// TwinCAT 3 PLC project LAP_2010_2_Transportwagen
// ProgramVersion: 3.1.4022.1
// libraries:
//   Tc2_Standard, * (Beckhoff Automation GmbH)
//   Tc2_System, * (Beckhoff Automation GmbH)
//   Tc2_Utilities, * (Beckhoff Automation GmbH)
//   Tc3_Module, * (Beckhoff Automation GmbH)
// project tree:
//   GVLs/ PlcCx9020.TcGVL, SimDI.TcGVL, SimDA.TcGVL, DigInput.TcGVL (not stored), DigOutput.TcGVL (not stored), AnalogInput.TcGVL (not stored), AnalogOutput.TcGVL (not stored), VersionsInfo.TcGVL (not stored)
//   / PlcTask.TcTTO (not stored)
//   POUs/ MAIN.TcPOU, Transportwagen.TcPOU
//   POUs/Privat/ AlleBitSetzen.TcPOU (not stored), BitLesen.TcPOU (not stored), DatenRangieren.TcPOU
// real-time tasks:
//   TASK PlcTask: cycle T#10ms, priority 20, ADS port 350
// motion (NC):
//   TASK NC-Task 1 SAF: cycle T#2ms, priority 4, ADS port 501
//   TASK NC-Task 1 SVB: cycle T#10ms, priority 8, ADS port 511
//   AXIS Axis 1 (id 1)
//     OtherSettings: AllowMotionCmdToSlave=true
//     encoder EncType=4
//       EncPara: MaxCount=#x0000ffff
//         Inc: RefSoftSyncMask=#x0000ffff
//     drive DrvType=24
//       Analog: ScaleFactorActTorque=0.1
//       TimeComp: TaskDelayCycles=1
//     controller CtrType=1
//       CtrPara: PriorControlFactor=1
//         Observer: BandWidth=20
//   AXIS Axis 2 (id 2)
//     OtherSettings: AllowMotionCmdToSlave=true
//     encoder EncType=4
//       EncPara: MaxCount=#x0000ffff
//         Inc: RefSoftSyncMask=#x0000ffff
//     drive DrvType=24
//       Analog: ScaleFactorActTorque=0.1
//       TimeComp: TaskDelayCycles=1
//     controller CtrType=1
//       CtrPara: PriorControlFactor=1
//         Observer: BandWidth=20
//   AXIS Axis 3 (id 3)
//     OtherSettings: AllowMotionCmdToSlave=true
//     encoder EncType=4
//       EncPara: MaxCount=#x0000ffff
//     drive DrvType=23
//       Analog: ScaleFactorActTorque=0.1
//       TimeComp: TaskDelayCycles=1
//     controller CtrType=1
//       CtrPara: PriorControlFactor=1
//         Observer: BandWidth=20
//   AXIS Axis 4 (id 4)
//     OtherSettings: AllowMotionCmdToSlave=true
//     encoder EncType=4
//       EncPara: MaxCount=#x0000ffff
//     drive DrvType=23
//       Analog: ScaleFactorActTorque=0.1
//       TimeComp: TaskDelayCycles=1
//     controller CtrType=1
//       CtrPara: PriorControlFactor=1
//         Observer: BandWidth=20
//   AXIS Axis 5 (id 5)
//     OtherSettings: AllowMotionCmdToSlave=true
//     encoder EncType=19
//       EncPara: MaxCount=#xffffffff
//     drive DrvType=16
//       DrvPara: MaxCount=#xffffffff
//         Analog: ScaleFactorActTorque=0.1
//         TimeComp: TaskDelayCycles=1
//     controller CtrType=1
//       CtrPara: PriorControlFactor=1
//         Observer: BandWidth=20
//   AXIS Axis 6 (id 6)
//     OtherSettings: AllowMotionCmdToSlave=true
//     encoder EncType=19
//       EncPara: MaxCount=#xffffffff
//     drive DrvType=16
//       DrvPara: MaxCount=#xffffffff
//         Analog: ScaleFactorActTorque=0.1
//         TimeComp: TaskDelayCycles=1
//     controller CtrType=1
//       CtrPara: PriorControlFactor=1
//         Observer: BandWidth=20
// I/O:
//   DEVICE Device 1 (EtherCAT), AmsNetId 192.168.0.200.2.1
//     Term 1 (EK1200) [EK1200-5000 EtherCAT Power supply (2A E-Bus)]
//       Term 2 (EL1809) [EL1809 16Ch. Dig. Input 24V, 3ms]
//       Term 3 (EL1809) [EL1809 16Ch. Dig. Input 24V, 3ms]
//       Term 4 (EL2809) [EL2809 16Ch. Dig. Output 24V, 0.5A]
//       Term 5 (EL2809) [EL2809 16Ch. Dig. Output 24V, 0.5A]
//       Term 6 (EL3064) [EL3064 4Ch. Ana. Input 0-10V]
//       Term 7 (EL4034) [EL4034 4Ch. Ana. Output +/-10V, 12bit]
//       Term 8 (EL7031) [EL7031 1Ch. Stepper motor output stage (24V, 1.5A)]
//       Term 9 (EL7031) [EL7031 1Ch. Stepper motor output stage (24V, 1.5A)]
//       Term 10 (EL7332) [EL7332 2Ch. DC motor output stage (24V, 1.5A)]
//       Term 11 (EL7201-0010) [EL7201-0010 1Ch. MDP742 Servo motor output stage with OCT (50V, 4A)]
//       Term 12 (EL7201-0010) [EL7201-0010 1Ch. MDP742 Servo motor output stage with OCT (50V, 4A)]
//       Term 26 (EL6090) [EL6090 Display terminal]
//       Term 27 (EK1110) [EK1110 EtherCAT extension]
// variable links:
//   NC-Task 1 SAF/Axes/Axis 1 <-> Device 1 (EtherCAT)/Term 1 (EK1200)/Term 8 (EL7031)
//     Drive/Inputs/In/nState1 @bit 3 <-> STM Status/Status/Error
//     Drive/Inputs/In/nState1 @bit 5 <-> STM Status/Status/Moving negative
//     Drive/Inputs/In/nState1 @bit 4 <-> STM Status/Status/Moving positive
//     Drive/Inputs/In/nState1 @bit 1 <-> STM Status/Status/Ready
//     Drive/Inputs/In/nState1 <-> STM Status/Status/Ready to enable
//     Drive/Inputs/In/nState1 @bit 6 <-> STM Status/Status/Torque reduced
//     Drive/Inputs/In/nState1 @bit 2 <-> STM Status/Status/Warning
//     Drive/Inputs/In/nState2 @bit 3 <-> STM Status/Status/Digital input 1
//     Drive/Inputs/In/nState2 @bit 4 <-> STM Status/Status/Digital input 2
//     Drive/Inputs/In/nState2 @bit 5 <-> STM Status/Status/Sync error
//     Drive/Inputs/In/nState2 @bit 7 <-> STM Status/Status/TxPDO Toggle
//     Drive/Inputs/In/nState4 @bit 1 <-> WcState/InputToggle
//     Drive/Inputs/In/nState4 <-> WcState/WcState
//     Drive/Outputs/Out/nCtrl1 <-> STM Control/Control/Enable
//     Drive/Outputs/Out/nCtrl1 @bit 2 <-> STM Control/Control/Reduce torque
//     Drive/Outputs/Out/nCtrl1 @bit 1 <-> STM Control/Control/Reset
//     Drive/Outputs/Out/nDataOut2[0] <-> STM Velocity/Velocity
//     Enc/Inputs/In/nDataIn1[0] <-> ENC Status compact/Counter value
//     Enc/Inputs/In/nDataIn2[0] <-> ENC Status compact/Latch value
//     Enc/Inputs/In/nState1 @bit 4 <-> ENC Status compact/Status/Counter overflow
//     Enc/Inputs/In/nState1 @bit 3 <-> ENC Status compact/Status/Counter underflow
//     Enc/Inputs/In/nState1 @bit 1 <-> ENC Status compact/Status/Latch extern valid
//     Enc/Inputs/In/nState1 @bit 2 <-> ENC Status compact/Status/Set counter done
//     Enc/Inputs/In/nState2 @bit 4 <-> ENC Status compact/Status/Status of extern latch
//     Enc/Inputs/In/nState2 @bit 5 <-> ENC Status compact/Status/Sync error
//     Enc/Inputs/In/nState2 @bit 7 <-> ENC Status compact/Status/TxPDO Toggle
//     Enc/Inputs/In/nState4 @bit 1 <-> WcState/InputToggle
//     Enc/Inputs/In/nState4 <-> WcState/WcState
//     Enc/Outputs/Out/nCtrl1 @bit 3 <-> ENC Control compact/Control/Enable latch extern on negative edge
//     Enc/Outputs/Out/nCtrl1 @bit 1 <-> ENC Control compact/Control/Enable latch extern on positive edge
//     Enc/Outputs/Out/nCtrl1 @bit 2 <-> ENC Control compact/Control/Set counter
//     Enc/Outputs/Out/nDataOut1[0] <-> ENC Control compact/Set counter value
//   NC-Task 1 SAF/Axes/Axis 2 <-> Device 1 (EtherCAT)/Term 1 (EK1200)/Term 9 (EL7031)
//     Drive/Inputs/In/nState1 @bit 3 <-> STM Status/Status/Error
//     Drive/Inputs/In/nState1 @bit 5 <-> STM Status/Status/Moving negative
//     Drive/Inputs/In/nState1 @bit 4 <-> STM Status/Status/Moving positive
//     Drive/Inputs/In/nState1 @bit 1 <-> STM Status/Status/Ready
//     Drive/Inputs/In/nState1 <-> STM Status/Status/Ready to enable
//     Drive/Inputs/In/nState1 @bit 6 <-> STM Status/Status/Torque reduced
//     Drive/Inputs/In/nState1 @bit 2 <-> STM Status/Status/Warning
//     Drive/Inputs/In/nState2 @bit 3 <-> STM Status/Status/Digital input 1
//     Drive/Inputs/In/nState2 @bit 4 <-> STM Status/Status/Digital input 2
//     Drive/Inputs/In/nState2 @bit 5 <-> STM Status/Status/Sync error
//     Drive/Inputs/In/nState2 @bit 7 <-> STM Status/Status/TxPDO Toggle
//     Drive/Inputs/In/nState4 @bit 1 <-> WcState/InputToggle
//     Drive/Inputs/In/nState4 <-> WcState/WcState
//     Drive/Outputs/Out/nCtrl1 <-> STM Control/Control/Enable
//     Drive/Outputs/Out/nCtrl1 @bit 2 <-> STM Control/Control/Reduce torque
//     Drive/Outputs/Out/nCtrl1 @bit 1 <-> STM Control/Control/Reset
//     Drive/Outputs/Out/nDataOut2[0] <-> STM Velocity/Velocity
//     Enc/Inputs/In/nDataIn1[0] <-> ENC Status compact/Counter value
//     Enc/Inputs/In/nDataIn2[0] <-> ENC Status compact/Latch value
//     Enc/Inputs/In/nState1 @bit 4 <-> ENC Status compact/Status/Counter overflow
//     Enc/Inputs/In/nState1 @bit 3 <-> ENC Status compact/Status/Counter underflow
//     Enc/Inputs/In/nState1 @bit 1 <-> ENC Status compact/Status/Latch extern valid
//     Enc/Inputs/In/nState1 @bit 2 <-> ENC Status compact/Status/Set counter done
//     Enc/Inputs/In/nState2 @bit 4 <-> ENC Status compact/Status/Status of extern latch
//     Enc/Inputs/In/nState2 @bit 5 <-> ENC Status compact/Status/Sync error
//     Enc/Inputs/In/nState2 @bit 7 <-> ENC Status compact/Status/TxPDO Toggle
//     Enc/Inputs/In/nState4 @bit 1 <-> WcState/InputToggle
//     Enc/Inputs/In/nState4 <-> WcState/WcState
//     Enc/Outputs/Out/nCtrl1 @bit 3 <-> ENC Control compact/Control/Enable latch extern on negative edge
//     Enc/Outputs/Out/nCtrl1 @bit 1 <-> ENC Control compact/Control/Enable latch extern on positive edge
//     Enc/Outputs/Out/nCtrl1 @bit 2 <-> ENC Control compact/Control/Set counter
//     Enc/Outputs/Out/nDataOut1[0] <-> ENC Control compact/Set counter value
//   NC-Task 1 SAF/Axes/Axis 3 <-> Device 1 (EtherCAT)/Term 1 (EK1200)/Term 10 (EL7332)
//     Drive/Inputs/In/nState1 @bit 3 <-> DCM Status Channel 1/Status/Error
//     Drive/Inputs/In/nState1 @bit 5 <-> DCM Status Channel 1/Status/Moving negative
//     Drive/Inputs/In/nState1 @bit 4 <-> DCM Status Channel 1/Status/Moving positive
//     Drive/Inputs/In/nState1 @bit 1 <-> DCM Status Channel 1/Status/Ready
//     Drive/Inputs/In/nState1 <-> DCM Status Channel 1/Status/Ready to enable
//     Drive/Inputs/In/nState1 @bit 6 <-> DCM Status Channel 1/Status/Torque reduced
//     Drive/Inputs/In/nState1 @bit 2 <-> DCM Status Channel 1/Status/Warning
//     Drive/Inputs/In/nState2 @bit 3 <-> DCM Status Channel 1/Status/Digital input 1
//     Drive/Inputs/In/nState2 @bit 4 <-> DCM Status Channel 1/Status/Digital input 2
//     Drive/Inputs/In/nState2 @bit 5 <-> DCM Status Channel 1/Status/Sync error
//     Drive/Inputs/In/nState2 @bit 7 <-> DCM Status Channel 1/Status/TxPDO Toggle
//     Drive/Inputs/In/nState4 @bit 1 <-> WcState/InputToggle
//     Drive/Inputs/In/nState4 <-> WcState/WcState
//     Drive/Outputs/Out/nCtrl1 <-> DCM Control Channel 1/Control/Enable
//     Drive/Outputs/Out/nCtrl1 @bit 2 <-> DCM Control Channel 1/Control/Reduce torque
//     Drive/Outputs/Out/nCtrl1 @bit 1 <-> DCM Control Channel 1/Control/Reset
//     Drive/Outputs/Out/nDataOut2[0] <-> DCM Velocity Channel 1/Velocity
//   NC-Task 1 SAF/Axes/Axis 4 <-> Device 1 (EtherCAT)/Term 1 (EK1200)/Term 10 (EL7332)
//     Drive/Inputs/In/nState1 @bit 3 <-> DCM Status Channel 2/Status/Error
//     Drive/Inputs/In/nState1 @bit 5 <-> DCM Status Channel 2/Status/Moving negative
//     Drive/Inputs/In/nState1 @bit 4 <-> DCM Status Channel 2/Status/Moving positive
//     Drive/Inputs/In/nState1 @bit 1 <-> DCM Status Channel 2/Status/Ready
//     Drive/Inputs/In/nState1 <-> DCM Status Channel 2/Status/Ready to enable
//     Drive/Inputs/In/nState1 @bit 6 <-> DCM Status Channel 2/Status/Torque reduced
//     Drive/Inputs/In/nState1 @bit 2 <-> DCM Status Channel 2/Status/Warning
//     Drive/Inputs/In/nState2 @bit 3 <-> DCM Status Channel 2/Status/Digital input 1
//     Drive/Inputs/In/nState2 @bit 4 <-> DCM Status Channel 2/Status/Digital input 2
//     Drive/Inputs/In/nState2 @bit 5 <-> DCM Status Channel 2/Status/Sync error
//     Drive/Inputs/In/nState2 @bit 7 <-> DCM Status Channel 2/Status/TxPDO Toggle
//     Drive/Inputs/In/nState4 @bit 1 <-> WcState/InputToggle
//     Drive/Inputs/In/nState4 <-> WcState/WcState
//     Drive/Outputs/Out/nCtrl1 <-> DCM Control Channel 2/Control/Enable
//     Drive/Outputs/Out/nCtrl1 @bit 2 <-> DCM Control Channel 2/Control/Reduce torque
//     Drive/Outputs/Out/nCtrl1 @bit 1 <-> DCM Control Channel 2/Control/Reset
//     Drive/Outputs/Out/nDataOut2[0] <-> DCM Velocity Channel 2/Velocity
//   NC-Task 1 SAF/Axes/Axis 5 <-> Device 1 (EtherCAT)/Term 1 (EK1200)/Term 11 (EL7201-0010)
//     Drive/Inputs/In/nDcOutputTime <-> InfoData/DcOutputShift
//     Drive/Inputs/In/nState1 <-> DRV Statusword/Statusword
//     Drive/Inputs/In/nState2 <-> DRV Statusword/Statusword @bit 8
//     Drive/Inputs/In/nState4 @bit 1 <-> WcState/InputToggle
//     Drive/Inputs/In/nState4 <-> WcState/WcState
//     Drive/Outputs/Out/nCtrl1 <-> DRV Controlword/Controlword
//     Drive/Outputs/Out/nCtrl2 <-> DRV Controlword/Controlword @bit 8
//     Drive/Outputs/Out/nDataOut2 <-> DRV Target velocity/Target velocity
//     Enc/Inputs/In/nDataIn1 <-> FB Position/Position
//     Enc/Inputs/In/nDcInputTime <-> InfoData/DcInputShift
//     Enc/Inputs/In/nState4 @bit 1 <-> WcState/InputToggle
//     Enc/Inputs/In/nState4 <-> WcState/WcState
//   NC-Task 1 SAF/Axes/Axis 6 <-> Device 1 (EtherCAT)/Term 1 (EK1200)/Term 12 (EL7201-0010)
//     Drive/Inputs/In/nDcOutputTime <-> InfoData/DcOutputShift
//     Drive/Inputs/In/nState1 <-> DRV Statusword/Statusword
//     Drive/Inputs/In/nState2 <-> DRV Statusword/Statusword @bit 8
//     Drive/Inputs/In/nState4 @bit 1 <-> WcState/InputToggle
//     Drive/Inputs/In/nState4 <-> WcState/WcState
//     Drive/Outputs/Out/nCtrl1 <-> DRV Controlword/Controlword
//     Drive/Outputs/Out/nCtrl2 <-> DRV Controlword/Controlword @bit 8
//     Drive/Outputs/Out/nDataOut2 <-> DRV Target velocity/Target velocity
//     Enc/Inputs/In/nDataIn1 <-> FB Position/Position
//     Enc/Inputs/In/nDcInputTime <-> InfoData/DcInputShift
//     Enc/Inputs/In/nState4 @bit 1 <-> WcState/InputToggle
//     Enc/Inputs/In/nState4 <-> WcState/WcState
//   LAP_2010_2_Transportwagen/LAP_2010_2_Transportwagen Instance <-> Device 1 (EtherCAT)/Term 1 (EK1200)/Term 2 (EL1809)
//     PlcTask Inputs/PlcCx9020.DI_0_0 <-> Channel 1/Input
//     PlcTask Inputs/PlcCx9020.DI_0_1 <-> Channel 2/Input
//     PlcTask Inputs/PlcCx9020.DI_0_2 <-> Channel 3/Input
//     PlcTask Inputs/PlcCx9020.DI_0_3 <-> Channel 4/Input
//     PlcTask Inputs/PlcCx9020.DI_0_4 <-> Channel 5/Input
//     PlcTask Inputs/PlcCx9020.DI_0_5 <-> Channel 6/Input
//     PlcTask Inputs/PlcCx9020.DI_0_6 <-> Channel 7/Input
//     PlcTask Inputs/PlcCx9020.DI_0_7 <-> Channel 8/Input
//     PlcTask Inputs/PlcCx9020.DI_1_0 <-> Channel 9/Input
//     PlcTask Inputs/PlcCx9020.DI_1_1 <-> Channel 10/Input
//     PlcTask Inputs/PlcCx9020.DI_1_2 <-> Channel 11/Input
//     PlcTask Inputs/PlcCx9020.DI_1_3 <-> Channel 12/Input
//     PlcTask Inputs/PlcCx9020.DI_1_4 <-> Channel 13/Input
//     PlcTask Inputs/PlcCx9020.DI_1_5 <-> Channel 14/Input
//     PlcTask Inputs/PlcCx9020.DI_1_6 <-> Channel 15/Input
//     PlcTask Inputs/PlcCx9020.DI_1_7 <-> Channel 16/Input
//   LAP_2010_2_Transportwagen/LAP_2010_2_Transportwagen Instance <-> Device 1 (EtherCAT)/Term 1 (EK1200)/Term 3 (EL1809)
//     PlcTask Inputs/PlcCx9020.DI_2_0 <-> Channel 1/Input
//     PlcTask Inputs/PlcCx9020.DI_2_1 <-> Channel 2/Input
//     PlcTask Inputs/PlcCx9020.DI_2_2 <-> Channel 3/Input
//     PlcTask Inputs/PlcCx9020.DI_2_3 <-> Channel 4/Input
//     PlcTask Inputs/PlcCx9020.DI_2_4 <-> Channel 5/Input
//     PlcTask Inputs/PlcCx9020.DI_2_5 <-> Channel 6/Input
//     PlcTask Inputs/PlcCx9020.DI_2_6 <-> Channel 7/Input
//     PlcTask Inputs/PlcCx9020.DI_2_7 <-> Channel 8/Input
//     PlcTask Inputs/PlcCx9020.DI_3_0 <-> Channel 9/Input
//     PlcTask Inputs/PlcCx9020.DI_3_1 <-> Channel 10/Input
//     PlcTask Inputs/PlcCx9020.DI_3_2 <-> Channel 11/Input
//     PlcTask Inputs/PlcCx9020.DI_3_3 <-> Channel 12/Input
//     PlcTask Inputs/PlcCx9020.DI_3_4 <-> Channel 13/Input
//     PlcTask Inputs/PlcCx9020.DI_3_5 <-> Channel 14/Input
//     PlcTask Inputs/PlcCx9020.DI_3_6 <-> Channel 15/Input
//     PlcTask Inputs/PlcCx9020.DI_3_7 <-> Channel 16/Input
//   LAP_2010_2_Transportwagen/LAP_2010_2_Transportwagen Instance <-> Device 1 (EtherCAT)/Term 1 (EK1200)/Term 4 (EL2809)
//     PlcTask Outputs/PlcCx9020.DA_0_0 <-> Channel 1/Output
//     PlcTask Outputs/PlcCx9020.DA_0_1 <-> Channel 2/Output
//     PlcTask Outputs/PlcCx9020.DA_0_2 <-> Channel 3/Output
//     PlcTask Outputs/PlcCx9020.DA_0_3 <-> Channel 4/Output
//     PlcTask Outputs/PlcCx9020.DA_0_4 <-> Channel 5/Output
//     PlcTask Outputs/PlcCx9020.DA_0_5 <-> Channel 6/Output
//     PlcTask Outputs/PlcCx9020.DA_0_6 <-> Channel 7/Output
//     PlcTask Outputs/PlcCx9020.DA_0_7 <-> Channel 8/Output
//     PlcTask Outputs/PlcCx9020.DA_1_0 <-> Channel 9/Output
//     PlcTask Outputs/PlcCx9020.DA_1_1 <-> Channel 10/Output
//     PlcTask Outputs/PlcCx9020.DA_1_2 <-> Channel 11/Output
//     PlcTask Outputs/PlcCx9020.DA_1_3 <-> Channel 12/Output
//     PlcTask Outputs/PlcCx9020.DA_1_4 <-> Channel 13/Output
//     PlcTask Outputs/PlcCx9020.DA_1_5 <-> Channel 14/Output
//     PlcTask Outputs/PlcCx9020.DA_1_6 <-> Channel 15/Output
//     PlcTask Outputs/PlcCx9020.DA_1_7 <-> Channel 16/Output
//   LAP_2010_2_Transportwagen/LAP_2010_2_Transportwagen Instance <-> Device 1 (EtherCAT)/Term 1 (EK1200)/Term 5 (EL2809)
//     PlcTask Outputs/PlcCx9020.DA_2_0 <-> Channel 1/Output
//     PlcTask Outputs/PlcCx9020.DA_2_1 <-> Channel 2/Output
//     PlcTask Outputs/PlcCx9020.DA_2_2 <-> Channel 3/Output
//     PlcTask Outputs/PlcCx9020.DA_2_3 <-> Channel 4/Output
//     PlcTask Outputs/PlcCx9020.DA_2_4 <-> Channel 5/Output
//     PlcTask Outputs/PlcCx9020.DA_2_5 <-> Channel 6/Output
//     PlcTask Outputs/PlcCx9020.DA_2_6 <-> Channel 7/Output
//     PlcTask Outputs/PlcCx9020.DA_2_7 <-> Channel 8/Output
//     PlcTask Outputs/PlcCx9020.DA_3_0 <-> Channel 9/Output
//     PlcTask Outputs/PlcCx9020.DA_3_1 <-> Channel 10/Output
//     PlcTask Outputs/PlcCx9020.DA_3_2 <-> Channel 11/Output
//     PlcTask Outputs/PlcCx9020.DA_3_3 <-> Channel 12/Output
//     PlcTask Outputs/PlcCx9020.DA_3_4 <-> Channel 13/Output
//     PlcTask Outputs/PlcCx9020.DA_3_5 <-> Channel 14/Output
//     PlcTask Outputs/PlcCx9020.DA_3_6 <-> Channel 15/Output
//     PlcTask Outputs/PlcCx9020.DA_3_7 <-> Channel 16/Output
//   LAP_2010_2_Transportwagen/LAP_2010_2_Transportwagen Instance <-> Device 1 (EtherCAT)/Term 1 (EK1200)/Term 6 (EL3064)
//     PlcTask Inputs/PlcCx9020.AI_{0..3} <-> AI Standard Channel {1..4}/Value  (4 links)
//   LAP_2010_2_Transportwagen/LAP_2010_2_Transportwagen Instance <-> Device 1 (EtherCAT)/Term 1 (EK1200)/Term 7 (EL4034)
//     PlcTask Outputs/PlcCx9020.AA_{0..3} <-> AO Outputs Channel {1..4}/Analog output  (4 links)

// ---- GVLs/PlcCx9020.TcGVL
{attribute 'qualified_only'}
VAR_GLOBAL
	// dSub 25
	DI_0_0 AT %IX0.0: BOOL;
	DI_0_1 AT %IX0.1: BOOL;
	DI_0_2 AT %IX0.2: BOOL;
	DI_0_3 AT %IX0.3: BOOL;
	DI_0_4 AT %IX0.4: BOOL;
	DI_0_5 AT %IX0.5: BOOL;
	DI_0_6 AT %IX0.6: BOOL;
	DI_0_7 AT %IX0.7: BOOL;
	DI_1_0 AT %IX1.0: BOOL;
	DI_1_1 AT %IX1.1: BOOL;
	DI_1_2 AT %IX1.2: BOOL;
	DI_1_3 AT %IX1.3: BOOL;
	DI_1_4 AT %IX1.4: BOOL;
	DI_1_5 AT %IX1.5: BOOL;
	DI_1_6 AT %IX1.6: BOOL;
	DI_1_7 AT %IX1.7: BOOL;
	// Sicherheitsbuchsen
	DI_2_0 AT %IX2.0: BOOL;
	DI_2_1 AT %IX2.1: BOOL;
	DI_2_2 AT %IX2.2: BOOL;
	DI_2_3 AT %IX2.3: BOOL;
	DI_2_4 AT %IX2.4: BOOL;
	DI_2_5 AT %IX2.5: BOOL;
	DI_2_6 AT %IX2.6: BOOL;
	DI_2_7 AT %IX2.7: BOOL;
	DI_3_0 AT %IX3.0: BOOL;
	DI_3_1 AT %IX3.1: BOOL;
	DI_3_2 AT %IX3.2: BOOL;
	DI_3_3 AT %IX3.3: BOOL;
	DI_3_4 AT %IX3.4: BOOL;
	DI_3_5 AT %IX3.5: BOOL;
	DI_3_6 AT %IX3.6: BOOL;
	DI_3_7 AT %IX3.7: BOOL;
	DI AT %IB0: ARRAY[0..3] OF BYTE; 

	// dSub 25
	DA_0_0 AT %QX0.0: BOOL;
	DA_0_1 AT %QX0.1: BOOL;
	DA_0_2 AT %QX0.2: BOOL;
	DA_0_3 AT %QX0.3: BOOL;
	DA_0_4 AT %QX0.4: BOOL;
	DA_0_5 AT %QX0.5: BOOL;
	DA_0_6 AT %QX0.6: BOOL;
	DA_0_7 AT %QX0.7: BOOL;
	DA_1_0 AT %QX1.0: BOOL;
	DA_1_1 AT %QX1.1: BOOL;
	DA_1_2 AT %QX1.2: BOOL;
	DA_1_3 AT %QX1.3: BOOL;
	DA_1_4 AT %QX1.4: BOOL;
	DA_1_5 AT %QX1.5: BOOL;
	DA_1_6 AT %QX1.6: BOOL;
	DA_1_7 AT %QX1.7: BOOL;
	// Sicherheitsbuchsen
	DA_2_0 AT %QX2.0: BOOL;
	DA_2_1 AT %QX2.1: BOOL;
	DA_2_2 AT %QX2.2: BOOL;
	DA_2_3 AT %QX2.3: BOOL;
	DA_2_4 AT %QX2.4: BOOL;
	DA_2_5 AT %QX2.5: BOOL;
	DA_2_6 AT %QX2.6: BOOL;
	DA_2_7 AT %QX2.7: BOOL;
	DA_3_0 AT %QX3.0: BOOL;
	DA_3_1 AT %QX3.1: BOOL;
	DA_3_2 AT %QX3.2: BOOL;
	DA_3_3 AT %QX3.3: BOOL;
	DA_3_4 AT %QX3.4: BOOL;
	DA_3_5 AT %QX3.5: BOOL;
	DA_3_6 AT %QX3.6: BOOL;
	DA_3_7 AT %QX3.7: BOOL;
	DA AT %QB0: ARRAY[0..3] OF BYTE;
	
	// dSub 25
	AI_0 AT %IW10: INT;			// Analogeingang 0
	AI_1 AT %IW12: INT;			// Analogeingang 1
	
	// Sicherheitsbuchsen
	AI_2 AT %IW14: INT;			// Analogeingang 2
	AI_3 AT %IW16: INT;			// Analogeingang 3
	AI AT %IW10: ARRAY[0..7] OF BYTE;
	
	
	// dSub 25
	AA_0 AT %QW10: INT;			// Analogausgang 0	
	// Sicherheitsbuchsen
	AA_1 AT %QW12: INT;			// Analogausgang 1	
	AA_2 AT %QW14: INT;			// Analogausgang 2	
	AA_3 AT %QW16: INT;			// Analogausgang 3	
	AA AT %QW10: ARRAY[0..7] OF BYTE;
	 	
END_VAR

// ---- GVLs/SimDI.TcGVL
{attribute 'qualified_only'}
VAR_GLOBAL
		// Endschalter Links
	B1 : BOOL; 
	// Endschalter REchts
	B2: BOOL;
	// Thermorelais
	F1: BOOL;
	// Taster Start
	S1: BOOL;
	// Taster NotHalt
	S2: BOOL;
	// Taster Reset
	S3: BOOL;
END_VAR

// ---- GVLs/SimDA.TcGVL
{attribute 'qualified_only'}
VAR_GLOBAL
	// Meldeleuchte "Störung"
	P1: BOOL;
	// Motor Linkslauf
	Q1: BOOL;
	// Motor Rechtslauf
	Q2: BOOL;
END_VAR

// ---- POUs/MAIN.TcPOU
PROGRAM MAIN
VAR
	Transportwagen: Transportwagen;
END_VAR

DatenRangieren();
Transportwagen();

END_PROGRAM

// ---- POUs/Transportwagen.TcPOU
FUNCTION_BLOCK Transportwagen
VAR_INPUT
END_VAR
VAR_OUTPUT
END_VAR
VAR
END_VAR

SimDA.P1:= SimDI.S1;
SimDA.Q1:= SimDI.S2;
SimDA.Q2:= SimDI.S3;

END_FUNCTION_BLOCK

// ---- POUs/Privat/DatenRangieren.TcPOU
PROGRAM DatenRangieren
VAR	
	VersionsText: STRING := 'LAP 2010/2 Transportwagen V2.0';
END_VAR

VersionsInfo.Ver := MAXSTRING_TO_BYTEARR(VersionsText);

IF (VersionsInfo.Befehle = 2#0000_00001) THEN

	SimDI.B1 := BitLesen(DigInput.DI[0],0);
	SimDI.B2 := BitLesen(DigInput.DI[0],1);
	SimDI.F1 := BitLesen(DigInput.DI[0],2);
	SimDI.S1 := BitLesen(DigInput.DI[0],3);
	SimDI.S2 := BitLesen(DigInput.DI[0],4);
	SimDI.S3 := BitLesen(DigInput.DI[0],5);
	
	DigOutput.DA[0] := AlleBitSetzen(	SimDa.P1,	
										SimDa.Q1,
										SimDa.Q2,	
										FALSE, FALSE, FALSE,  FALSE, FALSE);
ELSE
	
	SimDI.B1 := PlcCx9020.DI_0_0;
	SimDI.B2 := PlcCx9020.DI_0_1;
	SimDI.F1 := PlcCx9020.DI_0_2;
	SimDI.S1 := PlcCx9020.DI_0_3;
	SimDI.S2 := PlcCx9020.DI_0_4;
	SimDI.S3 := PlcCx9020.DI_0_5;
	
	PlcCx9020.DA_0_0 := SimDa.P1;
	PlcCx9020.DA_0_1 := SimDa.Q1;
	PlcCx9020.DA_0_2 := SimDa.Q2;
END_IF;

END_PROGRAM
